TYPE ST_System_TF_Zustand :
STRUCT
	Temp_Rueckl_Wand_Ost_Sektor1	: REAL;
	Temp_Rueckl_Wand_Ost_Sektor2	: REAL;
	Temp_Rueckl_Wand_Ost_Sektor3	: REAL;
	Temp_Rueckl_Wand_West_Sektor1	: REAL;
	Temp_Rueckl_Wand_West_Sektor2	: REAL;
	Temp_Rueckl_Wand_West_Sektor3	: REAL;
	Temp_Rueckl_Decke_Ost_Sektor1	: REAL;
	Temp_Rueckl_Decke_Ost_Sektor2	: REAL;
	Temp_Rueckl_Decke_Ost_Sektor3	: REAL;
	Temp_Rueckl_Decke_West_Sektor1	: REAL;
	Temp_Rueckl_Decke_West_Sektor2	: REAL;
	Temp_Rueckl_Decke_West_Sektor3	: REAL;
	Temp_Rueckl_Aussen_Ost			: REAL;
	Temp_Rueckl_Aussen_West			: REAL;
	Temp_Halle_Sektor1				:REAL;
	Temp_Halle_Sektor2				:REAL;
	Temp_Halle_Sektor3				:REAL;
	Wetter_Temperatur				:REAL;
	Temperatur_Aussen_TF			:REAL;
END_STRUCT
END_TYPE

(* stored: Version 1.1.0.1, ProductVersion 3.1.4024.9
   DUT ST_System_TF_Zustand: Id {7a36041a-3ee5-481e-a265-f29e43ce0c24} *)
